TYPE (* A Structure with 8 BOOLS *)
  (* Version 1.0, 2024-02-21, Franz Höpfinger, HR Agrartechnik GmbH *)
  PACKAGE logiBUS::utils::conversion::types;
  ST08X : STRUCT
    X_00 : BOOL; (* BIT 00 *)
    X_01 : BOOL; (* BIT 01 *)
    X_02 : BOOL; (* BIT 02 *)
    X_03 : BOOL; (* BIT 03 *)
    X_04 : BOOL; (* BIT 04 *)
    X_05 : BOOL; (* BIT 05 *)
    X_06 : BOOL; (* BIT 06 *)
    X_07 : BOOL; (* BIT 07 *)
  END_STRUCT;
END_TYPE
